INTERFACE I_PositionalDrive

METHOD atHome : BOOL
VAR_INPUT
END_VAR
END_METHOD

METHOD getPosition : LREAL
VAR_INPUT
END_VAR
END_METHOD

METHOD getTargetPosition : BOOL
VAR_INPUT
END_VAR
END_METHOD

METHOD hasError : BOOL
VAR_INPUT
END_VAR
END_METHOD

METHOD ABSTRACT homingSequence : BOOL
VAR_INPUT
END_VAR
END_METHOD

METHOD isBusy : BOOL
VAR_INPUT
END_VAR
END_METHOD

METHOD moveAbsolute : BOOL
VAR_INPUT
	newTarget : LREAL; 
END_VAR
END_METHOD

METHOD moveContinuous : BOOL
VAR_INPUT
	direction : MC_Direction;
END_VAR
END_METHOD

METHOD moveRelative : BOOL
VAR_INPUT
	distance : LREAL;
END_VAR
END_METHOD

END_INTERFACE

(* stored: Version 1.1.0.1, ProductVersion 3.1.4024.11
   Itf I_PositionalDrive: Id {542dde8d-3f0e-453c-8c39-9501a69f7da7}
   Folder Get: Id {312928f4-e4fd-4a43-994e-49d55c8ad75e}
   Method atHome: Id {eb79cbaa-9840-473c-83ef-bcfe177ce337}
   Method getPosition: Id {d85f7d3d-8b37-4622-9561-52092a485cf7}
   Method getTargetPosition: Id {33274651-146f-4855-b696-ae10599720d9}
   Method hasError: Id {9a4146e6-aa6a-4065-94fa-09229cb75d8a}
   Method homingSequence: Id {12409806-842f-4cb2-b5fe-f4a55b9c747a}
   Method isBusy: Id {cc17c0d7-ee05-4f61-ac84-32d58b665e57}
   Method moveAbsolute: Id {2c02535f-adbe-4dfa-ac4b-ddfb412f57da}
   Method moveContinuous: Id {bf078701-f572-4316-9dc9-8b0c8ae473a7}
   Method moveRelative: Id {83781e94-128b-41f5-8391-03ac83176760} *)
